// SIMATIC S7-200 project (STEP 7-Micro/WIN), CPU 224XP REL 02.01

ORGANIZATION_BLOCK PRINCIPAL:OB1
TITLE=COMENTARIOS DEL PROGRAMA
BEGIN
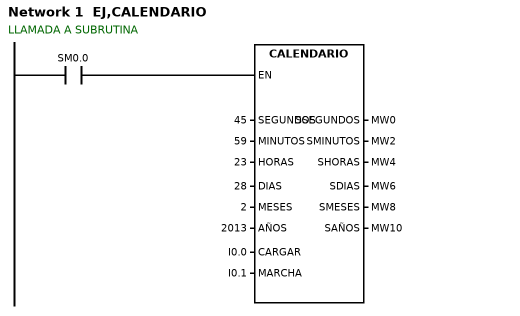
Network 1 // EJ,CALENDARIO
// LLAMADA A SUBRUTINA
LD     SM0.0
CALL   CALENDARIO:SBR0, 45, 59, 23, 28, 2, 2013, I0.0, I0.1, MW0, MW2, MW4, MW6, MW8, MW10
END_ORGANIZATION_BLOCK

SUBROUTINE_BLOCK CALENDARIO:SBR0
TITLE=COMENTARIOS DE LA SUBRUTINA
VAR_INPUT
SEGUNDOS:INT;	// LW0 
MINUTOS:INT;	// LW2 
HORAS:INT;	// LW4 
DIAS:INT;	// LW6 
MESES:INT;	// LW8 
AÑOS:INT;	// LW10 
CARGAR:BOOL;	// L12.0 
MARCHA:BOOL;	// L12.1 
END_VAR
VAR_OUTPUT
SSEGUNDOS:INT;	// LW13 
SMINUTOS:INT;	// LW15 
SHORAS:INT;	// LW17 
SDIAS:INT;	// LW19 
SMESES:INT;	// LW21 
SAÑOS:INT;	// LW23 
END_VAR
VAR
CSEGUNDOS:INT;	// LW25 
CMINUTOS:INT;	// LW27 
CHORAS:INT;	// LW29 
CDIAS:INT;	// LW31 
CMESES:INT;	// LW33 
CAÑOS:INT;	// LW35 
AUX30:BOOL;	// L37.0 
AUX28:BOOL;	// L37.1 
DRESULTADO:INT;	// LW38 
MRESULTADO:INT;	// LW40 
RESULTADO:INT;	// LW42 
BISIESTOAUX:BOOL;	// L44.0 
END_VAR
BEGIN
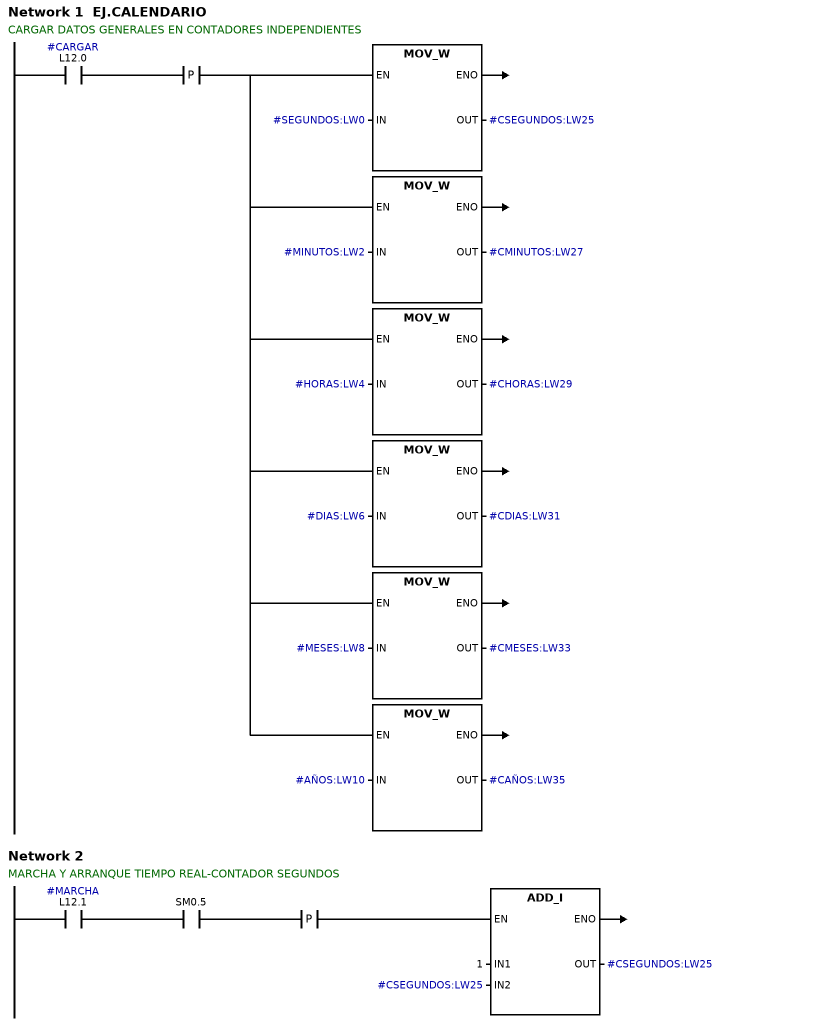
Network 1 // EJ.CALENDARIO
// CARGAR DATOS GENERALES EN CONTADORES INDEPENDIENTES
LD     #CARGAR:L12.0
EU
MOVW   #SEGUNDOS:LW0, #CSEGUNDOS:LW25
MOVW   #MINUTOS:LW2, #CMINUTOS:LW27
MOVW   #HORAS:LW4, #CHORAS:LW29
MOVW   #DIAS:LW6, #CDIAS:LW31
MOVW   #MESES:LW8, #CMESES:LW33
MOVW   #AÑOS:LW10, #CAÑOS:LW35
Network 2
// MARCHA Y ARRANQUE TIEMPO REAL-CONTADOR SEGUNDOS
LD     #MARCHA:L12.1
A      SM0.5
EU
+I     1, #CSEGUNDOS:LW25
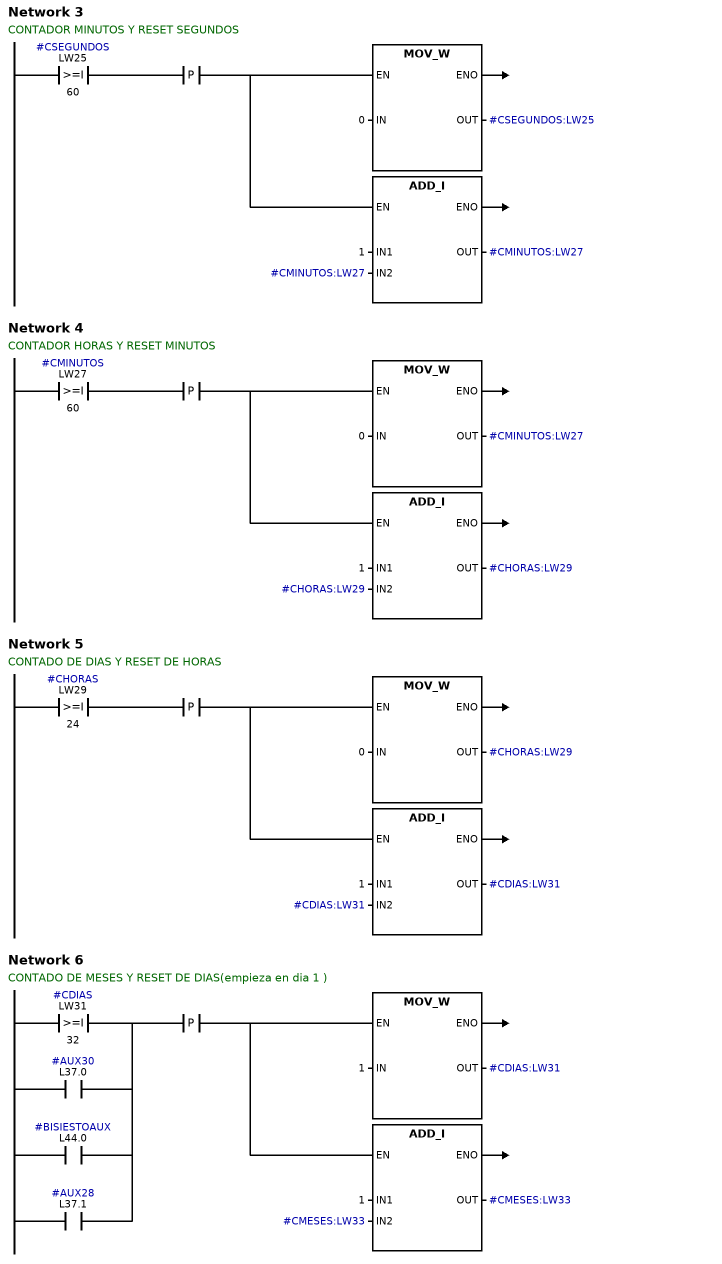
Network 3
// CONTADOR MINUTOS Y RESET SEGUNDOS
LDW>=  #CSEGUNDOS:LW25, 60
EU
MOVW   0, #CSEGUNDOS:LW25
+I     1, #CMINUTOS:LW27
Network 4
// CONTADOR HORAS Y RESET MINUTOS
LDW>=  #CMINUTOS:LW27, 60
EU
MOVW   0, #CMINUTOS:LW27
+I     1, #CHORAS:LW29
Network 5
// CONTADO DE DIAS Y RESET DE HORAS
LDW>=  #CHORAS:LW29, 24
EU
MOVW   0, #CHORAS:LW29
+I     1, #CDIAS:LW31
Network 6
// CONTADO DE MESES Y RESET DE DIAS(empieza en dia 1 )
LDW>=  #CDIAS:LW31, 32
O      #AUX30:L37.0
O      #BISIESTOAUX:L44.0
O      #AUX28:L37.1
EU
MOVW   1, #CDIAS:LW31
+I     1, #CMESES:LW33
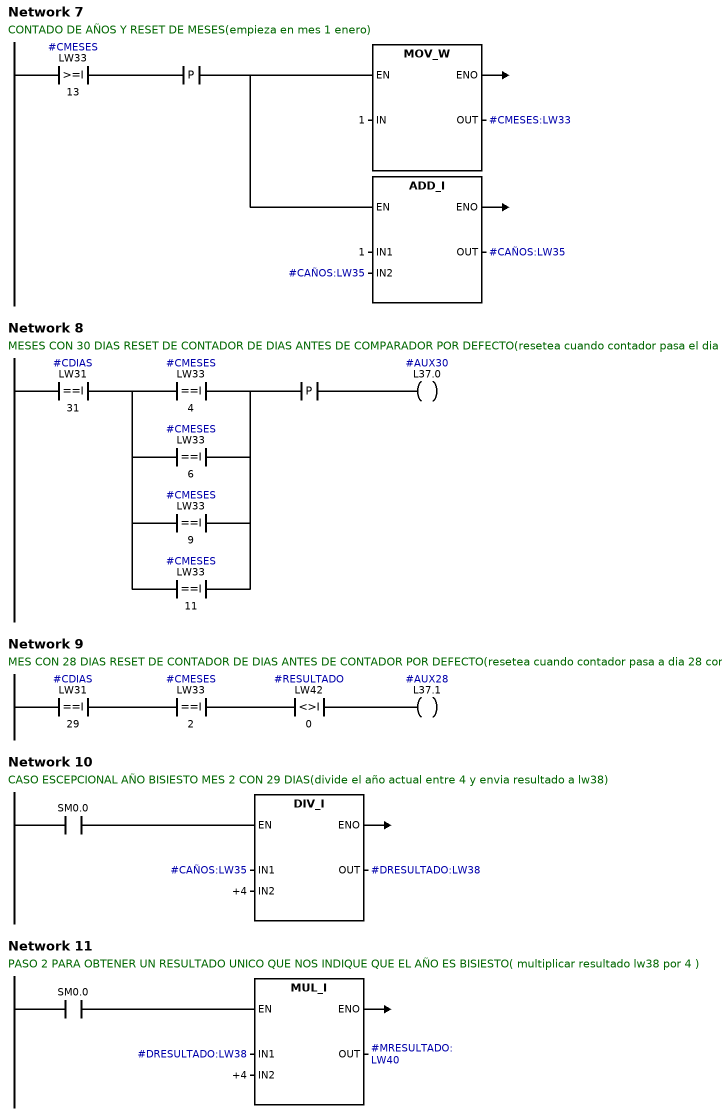
Network 7
// CONTADO DE AÑOS Y RESET DE MESES(empieza en mes 1 enero)
LDW>=  #CMESES:LW33, 13
EU
MOVW   1, #CMESES:LW33
+I     1, #CAÑOS:LW35
Network 8
// MESES CON 30 DIAS RESET DE CONTADOR DE DIAS ANTES DE COMPARADOR POR DEFECTO(resetea cuando contador pasa el dia 30 con sus 24 horas.es decie cunado marque 31)
LDW=   #CDIAS:LW31, 31
LDW=   #CMESES:LW33, 4
OW=    #CMESES:LW33, 6
OW=    #CMESES:LW33, 9
OW=    #CMESES:LW33, 11
ALD
EU
=      #AUX30:L37.0
Network 9
// MES CON 28 DIAS RESET DE CONTADOR DE DIAS ANTES DE CONTADOR POR DEFECTO(resetea cuando contador pasa a dia 28 con sus 24 horas,es decir cuando marque 29)
LDW=   #CDIAS:LW31, 29
AW=    #CMESES:LW33, 2
AW<>   #RESULTADO:LW42, 0
=      #AUX28:L37.1
Network 10
// CASO ESCEPCIONAL AÑO BISIESTO MES 2 CON 29 DIAS(divide el año actual entre 4 y envia resultado a lw38)
LD     SM0.0
MOVW   #CAÑOS:LW35, #DRESULTADO:LW38
/I     +4, #DRESULTADO:LW38
Network 11
// PASO 2 PARA OBTENER UN RESULTADO UNICO QUE NOS INDIQUE QUE EL AÑO ES BISIESTO( multiplicar resultado lw38 por 4 )
LD     SM0.0
MOVW   #DRESULTADO:LW38, #MRESULTADO:LW40
*I     +4, #MRESULTADO:LW40
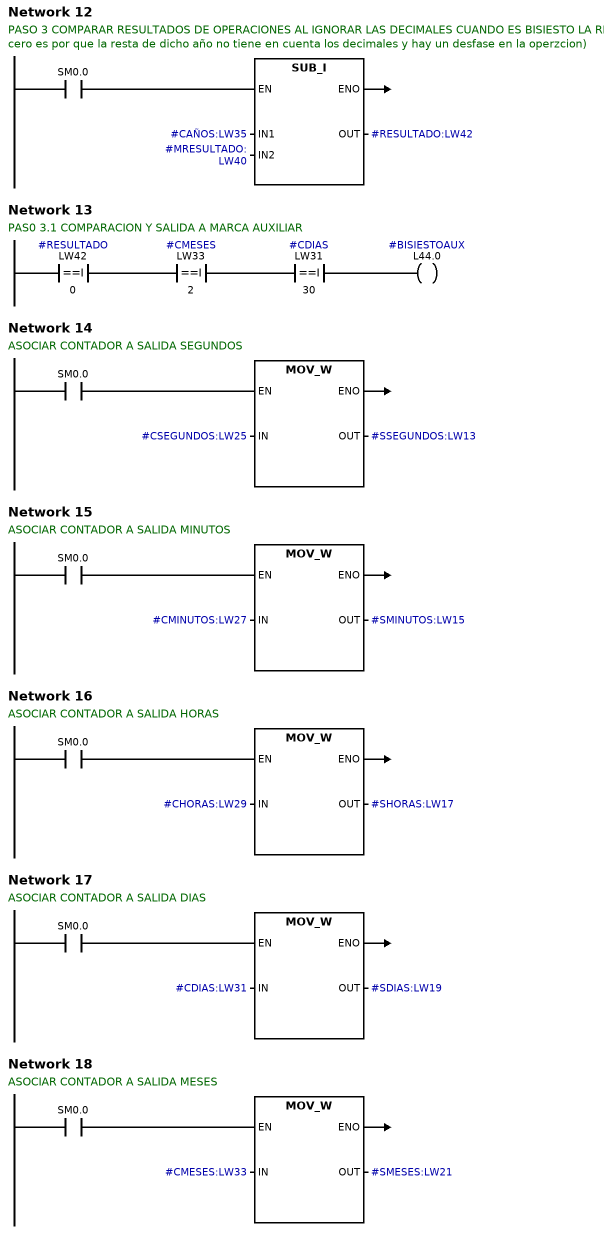
Network 12
// PASO 3 COMPARAR RESULTADOS DE OPERACIONES AL IGNORAR LAS DECIMALES CUANDO ES BISIESTO LA RESTA DEL AÑO  ANTES Y DESPUES DE LAS OPERACIONES SERA 0 (si la resta no es igual a cero es por que la resta de dicho año no tiene en cuenta los decimales y hay un desfase en la operzcion)
LD     SM0.0
MOVW   #CAÑOS:LW35, #RESULTADO:LW42
-I     #MRESULTADO:LW40, #RESULTADO:LW42
Network 13
// PAS0 3.1 COMPARACION Y SALIDA A MARCA AUXILIAR
LDW=   #RESULTADO:LW42, 0
AW=    #CMESES:LW33, 2
AW=    #CDIAS:LW31, 30
=      #BISIESTOAUX:L44.0
Network 14
// ASOCIAR CONTADOR A SALIDA SEGUNDOS
LD     SM0.0
MOVW   #CSEGUNDOS:LW25, #SSEGUNDOS:LW13
Network 15
// ASOCIAR CONTADOR A SALIDA MINUTOS
LD     SM0.0
MOVW   #CMINUTOS:LW27, #SMINUTOS:LW15
Network 16
// ASOCIAR CONTADOR A SALIDA HORAS
LD     SM0.0
MOVW   #CHORAS:LW29, #SHORAS:LW17
Network 17
// ASOCIAR CONTADOR A SALIDA DIAS 
LD     SM0.0
MOVW   #CDIAS:LW31, #SDIAS:LW19
Network 18
// ASOCIAR CONTADOR A SALIDA MESES 
LD     SM0.0
MOVW   #CMESES:LW33, #SMESES:LW21
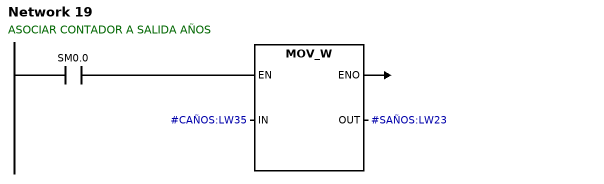
Network 19
// ASOCIAR CONTADOR A SALIDA AÑOS
LD     SM0.0
MOVW   #CAÑOS:LW35, #SAÑOS:LW23
END_SUBROUTINE_BLOCK
